DATA_BLOCK "KistlerPresser1_DB"
VAR
  ShaftID : Array[0..50] of Char;
  HousingID_1 : Array[0..50] of Char;
  HousingID_2 : Array[0..50] of Char;
  Shaft : String[48];
  spare : String[48];
END_VAR
BEGIN
END_DATA_BLOCK
